INTERFACE I_AdsAccess EXTENDS I_Base

PROPERTY AdsRW : I_AdsRW
GET
END_GET
SET
END_SET
END_PROPERTY

END_INTERFACE

(* stored: Version 1.1.0.1, ProductVersion 3.1.4026.18
   Itf I_AdsAccess: Id {28c023fc-e5c3-44ad-b222-07c7ba41bc96}
   Property AdsRW: Id {9f4bc844-73f3-4a77-8715-e73a39bb47ca}
   Get Get: Id {097d335d-ecac-4073-bb72-dfdff801f537}
   Set Set: Id {28c21864-eb82-454e-b7de-a961167d710f} *)
